(* PLC project actuator, TNI-Software ControlBuild 4.00.17 *)
(* stored: creationDateTime 2005-06-20T11:54:19-01:00 *)

FUNCTION_BLOCK cmd_equipment_library.actuator
  VAR_INPUT  (* CB.group=Modes CB.kind=inputVars *)
    autoMode : BOOL := false;  (* CB.libelle=Automatic mode *)
    manualMode : BOOL := false;  (* CB.libelle=Manual mode *)
  END_VAR
  VAR_INPUT  (* CB.group=Commands CB.kind=inputVars *)
    autoCloseCmd : BOOL := false;  (* CB.libelle=Automatic close command to the valve *)
    autoOpenCmd : BOOL := false;  (* CB.libelle=Automatic open command to the valve *)
  END_VAR
  VAR_INPUT  (* CB.group=Sensors CB.kind=inputVars *)
    closedSensorFB : BOOL := false;  (* CB.libelle=Closed sensor feedback *)
    openedSensorFB : BOOL := false;  (* CB.libelle=Opened sensor feedback *)
  END_VAR
  VAR_INPUT  (* CB.group=PushButtons CB.kind=inputVars *)
    closeValvePB : BOOL := false;  (* CB.libelle=Close valve pushbutton *)
    openValvePB : BOOL := false;  (* CB.libelle=Open valve pushbutton *)
  END_VAR
  VAR_INPUT  (* CB.kind=inputVars *)
    generalFault : BOOL := false;  (* CB.mnemonicPatternPropertyName=defGeneral<SY><NU> CB.libelle=General fault of the valve *)
  END_VAR
  VAR_OUTPUT  (* CB.group=Orders CB.kind=outputVars *)
    closeCmd : BOOL := false;  (* CB.mnemonicPatternPropertyName=closeCmd<SY><NU> CB.libelle=Close command to the valve *)
    openCmd : BOOL := false;  (* CB.mnemonicPatternPropertyName=openCmd<SY><NU> CB.libelle=Open command to the valve *)
  END_VAR

(* LD diagram, written out as Structured Text *)
1:
openCmd := (autoMode AND autoOpenCmd AND NOT autoCloseCmd OR manualMode AND openValvePB AND NOT closeValvePB) AND NOT openedSensorFB AND NOT generalFault;
2:
closeCmd := (autoMode AND autoCloseCmd AND NOT autoOpenCmd OR manualMode AND closeValvePB AND NOT openValvePB) AND NOT closedSensorFB AND NOT generalFault;
END_FUNCTION_BLOCK
